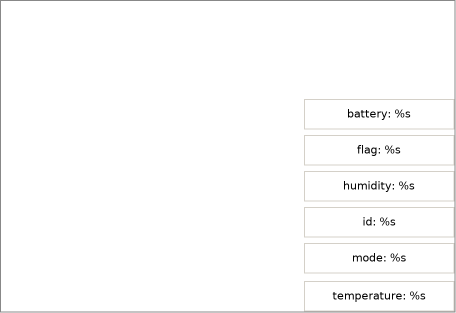
VISUALIZATION Visualization  // 456x313
    Textfield (304,99 150x30), "battery: %s", text variable: JSON_decode.mydata.battery
    Textfield (304,135 150x30), "flag: %s", text variable: JSON_decode.mydata.flag
    Textfield (304,171 150x30), "humidity: %s", text variable: JSON_decode.mydata.hum
    Textfield (304,207 150x30), "id: %s", text variable: JSON_decode.mydata.id
    Textfield (304,243 150x30), "mode: %s", text variable: JSON_decode.mydata.mode
    Textfield (304,281 150x30), "temperature: %s", text variable: JSON_decode.mydata.temp
END_VISUALIZATION

(* stored: Version 1.1.0.1, ProductVersion 3.1.4024.0
   Visu Visualization: Id {40e7b8ad-7c92-471a-9dda-938c13b63771} *)
